{attribute 'qualified_only'}
VAR_GLOBAL
	
//HMI
	



//Factory IO 
	//Inputs
		// MACH CNTR BUSY
			b_IN_0: BOOL;
		// MACH CNTR ERR
			b_IN_1: BOOL;
		// CONTAIN EMIT PE
			b_IN_2: BOOL;
		// BASE VISION SENS
			b_IN_3: BOOL;
		// INPUT CONV 1 PE
			b_IN_4: BOOL;
		// INPUT PICKUP PE
			b_IN_5: BOOL;
		// OUT DEP CONV PE
			b_IN_6: BOOL;
		// OUT CONV 1 PE
			b_IN_7: BOOL;
		// OUT CONV 2 PE
			b_IN_8: BOOL;
		// CRANE MOVE X
			b_IN_9: BOOL;
		// CRANE MOVE Z
			b_IN_10: BOOL;
		// CRANE LEFT LS
			b_IN_11: BOOL;
		// CRANE RIGHT LS
			b_IN_12: BOOL;
		// CRANE MID LS
			b_IN_13: BOOL;
		// UNUSED
			b_IN_14: BOOL;
		// UNUSED
			b_IN_15: BOOL;
		// UNUSED
			b_IN_64: BOOL;
	
	
		// Machining Center  Progress
			r_IN_0: WORD;
		//Light Array Emitter
			r_IN_1: WORD;
//Outputs
		// RAW MAT EMIT
			b_OUT_0: BOOL;
		// MACH LIDS
			b_OUT_1: BOOL;
		// CONTAIN CONV EMIT
			b_OUT_2: BOOL;
		// CONTAIN CONV MS
			b_OUT_3: BOOL := FALSE;
		// CONV PICK MS
			b_OUT_4: BOOL;
		// OUT DEP CONV MS
			b_OUT_5: BOOL;
		// OUT CONV 1 MS
			b_OUT_6: BOOL;
		// OUT CONV 2 MS
			b_OUT_7: BOOL;
		// OUT CONV REMOVE
			b_OUT_8: BOOL;
		// CRANE LIFT
			b_OUT_9: BOOL;
		// CRANE LEFT
			b_OUT_10: BOOL;
		// CRANE RIGHT
			b_OUT_11: BOOL;
		// INPUT CONV 1 MS
			b_OUT_12: BOOL;
		// CNC MACH RESET
			b_OUT_13: BOOL;
		// UNUSED
			b_OUT_14: BOOL;
		// UNUSED
			b_OUT_15: BOOL;
		// UNUSED
			b_OUT_16: BOOL;
		
		
		//Stacker Crane Target Position
			r_out_0: WORD;

END_VAR

(* stored: Version 1.1.0.1
   GVL FIO: Id {ab95a793-e106-4adf-a3e7-761095c7de4f} *)
